// =============================================================================
// Version_Recipe - 05_RecipeHandler.scl
// Recipe-based motion handler with pre-scan validation
// No string parsing - direct array access for maximum efficiency
// =============================================================================

// -----------------------------------------------------------------------------
// FB_RecipeLoader - Copy the selected recipe from LOAD memory into work memory
// DOC:
//  purpose: DB_RecipeProgram1..PROGRAM_COUNT live in load memory (UNLINKED) and cannot be
//           read by the program directly. This FB copies the selected one into
//           "DB_SelectedRecipe" using TWO sequential READ_DBL sub-reference
//           transfers -- .Header first, then .Lines. Never the whole-DB form;
//           see "TWO TRANSFERS, NOT ONE" below for what that cost on the machine.
//           Runs once per cycle start, in STATE_RECIPE_LOAD(11), before the
//           pre-scan -- the machine is stationary and nothing else is pending.
//  inputs:  Execute (rising edge), ProgramNo (1..PROGRAM_COUNT), Reset (level)
//  outputs: Done, Busy, Error + ErrorCode, LoadedProgram
//  design:  Program/docs/LOADMEM_COPY_ON_SELECT.md  (gate-tested 2026-08-04)
//
//  READ_DBL call form -- both of these cost a build if you get them wrong:
//    * READ_DBL is an INSTANCE-LESS system function (SFC 83 heritage). Declaring
//      it as a multi-instance gives "Data type READ_DBL is unknown".
//    * RET_VAL is the FUNCTION RETURN VALUE, not an output parameter. Passing
//      it as RET_VAL => x gives "The formal parameter 'RET_VAL' is invalid".
//
//  TWO TRANSFERS, NOT ONE (changed 2026-08-06 after a field failure).
//  The first version copied the WHOLE DB in one call (SRCBLK := "DB_RecipeProgramN").
//  On the machine that delivered the Header correctly and left Lines completely
//  zero, with no error anywhere -- a structured copy that matched the first
//  member and gave up on the second. Re-reading the gate-test results
//  (loadmem_gatetest/result.md) shows why it was never caught: whole-DB mode was
//  only ever proven at 350 lines / 4.3 KB, while the 12 KB / 1000-line case was
//  proven with the SUB-REFERENCE form (SRCBLK := "...".Lines). Production ran the
//  one combination -- whole DB at 12 KB -- that no test covered.
//  So: Header and Lines are now copied in two sequential calls, each in the exact
//  form the gate test passed. A length or type mismatch on Lines surfaces as a
//  non-zero RET_VAL instead of a silently empty buffer.
//
//  THE SPLIT WAS NOT ENOUGH (2026-08-13, second field failure, same signature).
//  The claim that a sub-reference copy "cannot half-succeed" was wrong. On the
//  machine the .Lines call again returned RET_VAL = 0 with BUSY = FALSE while the
//  array stayed zero -- pre-scan caught it as 16#0313. RET_VAL/BUSY report that the
//  instruction accepted and closed the job, not that 12 KB of flash arrived, and
//  the moment this FB left ST_WAIT_LINES it dropped REQ and abandoned whatever was
//  still in flight. PLCSIM never reproduced it (host RAM, copy done in one call).
//  ST_WAIT_LINES therefore no longer trusts BUSY alone: it VERIFIES the copy and
//  re-issues the transfer up to LINES_RETRY_MAX times before failing. Do not
//  "simplify" that check away -- it is the only thing standing between a silent
//  partial copy and a machined part.
//
//  WHY THE VERIFY PROBES THE WHOLE ARRAY AND NOT JUST THE END MARKER.
//  Same day, with a 999-line recipe: the operator found DB_SelectedRecipe zero up
//  to roughly line 900 and CORRECT after it. The copy is not all-or-nothing, it is
//  PARTIAL -- and the part that landed is where the END marker lives, so a
//  marker-only test would have passed that buffer and the machine would have run
//  ~900 zero lines (X=0, Z=0) with the HMI counting up. That is exactly what
//  happened before this check existed. Five sampled probes replaced the marker
//  test, and chunking replaced the samples: at CHUNK_LINES = 100 EVERY line of the
//  staging buffer is poisoned and checked, so coverage is complete rather than
//  statistical. The 38-line case is the same fault seen from the other end: there
//  the marker sits at index 37, in the region that did NOT land, so pre-scan
//  caught it as 16#0313.
//  ErrorPhase says what failed: 1 = Header, 2 = chunk transfer, 3 = chunk verify.
//
//  WHAT THE VERIFY STILL CANNOT SEE, AND THE CHECKSUM (2026-08-14).
//  Poisoning proves every line was WRITTEN. It says nothing about whether the
//  right data arrived: a stale flash image, chunks reassembled at the wrong
//  stride, or a Header paired with another export's Lines all pass it, because
//  in every one of those cases all 1000 lines are written. So the loader now
//  folds an order-sensitive checksum over CMD + Param + F into ST_CHUNK_COPY
//  (the loop that already walks every line -- four adds per line, no second
//  pass) and compares it with Header.Checksum after the last chunk. Mismatch =
//  16#0316, ErrorPhase 4. Header.ProvidesChecksum = FALSE skips the check so
//  pre-2026-08-14 exports still load; that is deliberate, not a hole to close.
//  X and Z are NOT in the sum -- float32 on the CPU against float64 in the CAM
//  would eventually disagree on a VALID recipe, and an alarm that cries wolf is
//  worse than no alarm. Spec both sides build to:
//  Program/docs/letter_spinningcam_recipe_checksum.md
//
//  READING A FAILED LOAD (2026-08-14). ST_LATCH poisons every CMD in
//  DB_SelectedRecipe.Lines with 16#FF before the first transfer, so after a
//  failure the buffer says which chunks got in: 16#FF = never copied, 0 = copied
//  and the source is zero there, valid CMD = copied intact. ErrorChunk names the
//  chunk that ran out of retries; the poison shows what surrounds it.
//
//  THE SELECTION LATCH -- the one genuinely dangerous thing in this block.
//  READ_DBL is asynchronous and spans several scans with REQ held. SRCBLK is a
//  VARIANT and the S7-1200 cannot index a DB dynamically, so the source is
//  chosen by a CASE. If that CASE branch changed mid-transfer, the buffer would
//  receive the front of one recipe and the tail of another -- with RET_VAL = 0
//  and no error anywhere. The operator would machine a part that exists in no
//  recipe. Hence #selLatched: the branch is frozen at ST_LATCH and the live
//  ProgramNo input is ignored until the transfer completes.
//
//  Reset path: REQ is derived from the state EVERY scan and is never latched
//  independently, so there is no way for a transfer to stay in flight across a
//  reset, an E-Stop or an error acknowledge.
// -----------------------------------------------------------------------------
FUNCTION_BLOCK "FB_RecipeLoader"
{ S7_Optimized_Access := 'TRUE' }
VERSION : 0.3
    VAR_INPUT
        Execute   : Bool;           // Rising edge starts the copy
        ProgramNo : Int;            // 1..PROGRAM_COUNT -- which recipe to load
        Reset     : Bool;           // Level: abort, clear error, invalidate buffer
    END_VAR
    VAR_OUTPUT
        Done          : Bool;       // Copy complete AND verified, DB_SelectedRecipe is valid
        Busy          : Bool;       // Transfer in flight
        Error         : Bool;       // Copy failed -- FB_Process raises 16#0312 or 16#0314
        ErrorCode     : Word;       // READ_DBL RET_VAL, latched. Two sentinels that are
                                    // NOT RET_VAL values: 16#FFFF = watchdog timeout,
                                    // 16#0314 = a chunk never arrived intact
        ErrorPhase    : Int;        // 1 = Header transfer, 2 = chunk transfer (RET_VAL),
                                    // 3 = chunk verify (RET_VAL said OK, data did not arrive),
                                    // 4 = checksum mismatch (it all arrived, but it is not
                                    //     the recipe the CAM exported)
        ErrorChunk    : Int;        // Which chunk failed (1..CHUNK_COUNT), 0 = Header or
                                    // the assembled-buffer end-marker check
        RetryTotal    : Int;        // Re-issued transfers across the WHOLE load, cleared
                                    // at ST_LATCH. This is the margin gauge: a load that
                                    // succeeds with RetryTotal = 0 is comfortable; one
                                    // that succeeds with RetryTotal > 0 got there on
                                    // second attempts and CHUNK_LINES is too close to
                                    // whatever this CPU can actually deliver. Watch it on
                                    // the first hardware run -- a clean Done tells you
                                    // nothing on its own.
        LoadedProgram : Int;        // Which recipe is in the buffer (0 = none/invalid)
        ChecksumCalc  : UDInt;      // What WE computed over the reassembled buffer. On a
                                    // 16#0316 this is the number to compare against
                                    // DB_SelectedRecipe.Header.Checksum by hand -- and to
                                    // quote to the CAM developer, because one of the two
                                    // implementations is wrong and the pair says which.
        ChecksumOK    : Bool;       // TRUE = checked and matched. FALSE also means "the
                                    // recipe carries no checksum", so it is NOT a fault
                                    // indicator on its own -- read it with ProvidesChecksum.
    END_VAR
    VAR
        // READ_DBL is NOT declared here -- see the note above.
        tonWatch    : TON;          // Hang watchdog (RecipeLoadTimeout), per transfer
        state       : Int;          // see the ST_* constants below
        selLatched  : Int := 1;     // Frozen program number for the whole load.
                                    // Never cleared: keeps the instruction being
                                    // called with REQ=FALSE so it resets cleanly.
        chunkPhase  : Int;          // 0 = Header is the live call, 1..CHUNK_COUNT = that
                                    // chunk. Latched like selLatched: only ever changed
                                    // where REQ is already low, never mid-transfer.
        chunkRetry  : Int;          // Attempts already re-issued for the CURRENT chunk
        reqActive   : Bool;         // REQ level, derived from state every scan
        busyRaw     : Bool;         // READ_DBL BUSY
        retValRaw   : Int;          // READ_DBL return value (raw, every scan)
        chunkOK     : Bool;         // every line of the staging buffer came back written
        hdrLines    : Int;          // Header.LineCount, latched at ST_HDR_SETTLE. Used by
                                    // the checksum fold and the END-marker check, so it is
                                    // read ONCE from the Header and not re-read per chunk.
        dstBase     : Int;          // first DB_SelectedRecipe index of the current chunk
        sumA        : UDInt;        // checksum accumulator: running line sum
        sumB        : UDInt;        // checksum accumulator: sum of sumA -> order-sensitive
        prevExecute : Bool;
        rtExecute   : Bool;
    END_VAR
    VAR_TEMP
        i           : Int;          // loop index (poison / verify / copy)
        gLine       : Int;          // global recipe line index during the copy
    END_VAR
    CONST
        ST_IDLE        : Int := 0;
        ST_LATCH       : Int := 10;
        ST_REQ_HDR     : Int := 20;  // Header transfer
        ST_WAIT_HDR    : Int := 30;
        ST_HDR_SETTLE  : Int := 35;  // One scan with REQ low so the Header call sees
                                     // its job closed before the CASE switches
        ST_CHUNK_PREP  : Int := 38;  // REQ low: poison the staging buffer, then request.
                                     // Also the settle scan BETWEEN chunks and the
                                     // re-poison step before a retry.
        ST_REQ_CHUNK   : Int := 40;
        ST_WAIT_CHUNK  : Int := 50;
        ST_CHUNK_COPY  : Int := 57;  // staging -> DB_SelectedRecipe (work memory, sync)
        ST_DONE        : Int := 60;
        ST_ERROR       : Int := 90;
        CHUNK_RETRY_MAX : Int := 3;  // re-issues per chunk before 16#0314. Each attempt
                                     // is bounded by RecipeLoadTimeout.
        CMD_PROGRAM_END : Int := 99; // Mandatory last-line marker (PLC_Recipe_Format_Spec.md)
        POISON_CMD     : Int := 255; // 16#FF -- no recipe CMD can be this value
        // Chunk geometry. COUPLED to tools/gen_recipe_slots.py (CHUNK_LINES /
        // CHUNK_COUNT) and to the DB_RecipeProgram*.Lines1..N declarations it
        // emits. Change them together or the transfers go out of step.
        // <<< GENERATED:CHUNK_GEOMETRY -- do not hand-edit; run tools/gen_recipe_slots.py >>>
        CHUNK_LINES    : Int := 100;
        CHUNK_COUNT    : Int := 8;
        LINES_MAX      : Int := 800; // = CHUNK_LINES * CHUNK_COUNT, and the bound of
                                      // DB_SelectedRecipe.Lines + the pre-scan guard
        // <<< END GENERATED:CHUNK_GEOMETRY >>>
        // <<< GENERATED:PROGRAM_COUNT -- do not hand-edit; run tools/gen_recipe_slots.py >>>
        PROGRAM_COUNT : Int := 10;  // Slot count. Generated -- must match the DB_RecipeProgram* count.
        // <<< END GENERATED:PROGRAM_COUNT >>>
    END_CONST
BEGIN
    // -------------------------------------------------------------------------
    // Rising edge on Execute
    // -------------------------------------------------------------------------
    #rtExecute := #Execute AND NOT #prevExecute;
    #prevExecute := #Execute;

    // -------------------------------------------------------------------------
    // Reset -- always honoured. Drives REQ low via the state on the next line.
    // -------------------------------------------------------------------------
    IF #Reset THEN
        #state := ST_IDLE;
        #Done := FALSE;
        #Error := FALSE;
        #ErrorCode := 16#0000;
        #ErrorPhase := 0;
        #ErrorChunk := 0;
        #chunkPhase := 0;           // idle on the Header branch, REQ low
        #chunkRetry := 0;
        #RetryTotal := 0;
        #LoadedProgram := 0;        // Buffer is no longer trusted -> forces a re-load
        #ChecksumCalc := 0;
        #ChecksumOK := FALSE;
    END_IF;

    // -------------------------------------------------------------------------
    // REQ is derived from state EVERY SCAN -- never latched on its own.
    // ST_CHUNK_PREP is deliberately excluded: that is the scan where the previous
    // job is closed, the staging buffer is poisoned and the watchdog resets.
    // -------------------------------------------------------------------------
    #reqActive := (#state = ST_REQ_HDR) OR (#state = ST_WAIT_HDR)
                  OR (#state = ST_REQ_CHUNK) OR (#state = ST_WAIT_CHUNK);

    // -------------------------------------------------------------------------
    // THE READ_DBL CALL BLOCK
    // Outer CASE = which recipe (#selLatched), inner CASE = which transfer
    // (#chunkPhase: 0 = Header, 1..CHUNK_COUNT = Lines chunks). Exactly ONE call
    // executes per scan. Both selectors are latched, never the live inputs.
    // -------------------------------------------------------------------------
    // <<< GENERATED:LOADER_CASE -- do not hand-edit; run tools/gen_recipe_slots.py >>>
    CASE #selLatched OF
        1:  CASE #chunkPhase OF
                0: #retValRaw := READ_DBL(REQ := #reqActive, SRCBLK := "DB_RecipeProgram1".Header,
                                           BUSY => #busyRaw, DSTBLK := "DB_SelectedRecipe".Header);
                1: #retValRaw := READ_DBL(REQ := #reqActive, SRCBLK := "DB_RecipeProgram1".Lines1,
                                           BUSY => #busyRaw, DSTBLK := "DB_RecipeChunk".Lines);
                2: #retValRaw := READ_DBL(REQ := #reqActive, SRCBLK := "DB_RecipeProgram1".Lines2,
                                           BUSY => #busyRaw, DSTBLK := "DB_RecipeChunk".Lines);
                3: #retValRaw := READ_DBL(REQ := #reqActive, SRCBLK := "DB_RecipeProgram1".Lines3,
                                           BUSY => #busyRaw, DSTBLK := "DB_RecipeChunk".Lines);
                4: #retValRaw := READ_DBL(REQ := #reqActive, SRCBLK := "DB_RecipeProgram1".Lines4,
                                           BUSY => #busyRaw, DSTBLK := "DB_RecipeChunk".Lines);
                5: #retValRaw := READ_DBL(REQ := #reqActive, SRCBLK := "DB_RecipeProgram1".Lines5,
                                           BUSY => #busyRaw, DSTBLK := "DB_RecipeChunk".Lines);
                6: #retValRaw := READ_DBL(REQ := #reqActive, SRCBLK := "DB_RecipeProgram1".Lines6,
                                           BUSY => #busyRaw, DSTBLK := "DB_RecipeChunk".Lines);
                7: #retValRaw := READ_DBL(REQ := #reqActive, SRCBLK := "DB_RecipeProgram1".Lines7,
                                           BUSY => #busyRaw, DSTBLK := "DB_RecipeChunk".Lines);
                8: #retValRaw := READ_DBL(REQ := #reqActive, SRCBLK := "DB_RecipeProgram1".Lines8,
                                           BUSY => #busyRaw, DSTBLK := "DB_RecipeChunk".Lines);
            END_CASE;
        2:  CASE #chunkPhase OF
                0: #retValRaw := READ_DBL(REQ := #reqActive, SRCBLK := "DB_RecipeProgram2".Header,
                                           BUSY => #busyRaw, DSTBLK := "DB_SelectedRecipe".Header);
                1: #retValRaw := READ_DBL(REQ := #reqActive, SRCBLK := "DB_RecipeProgram2".Lines1,
                                           BUSY => #busyRaw, DSTBLK := "DB_RecipeChunk".Lines);
                2: #retValRaw := READ_DBL(REQ := #reqActive, SRCBLK := "DB_RecipeProgram2".Lines2,
                                           BUSY => #busyRaw, DSTBLK := "DB_RecipeChunk".Lines);
                3: #retValRaw := READ_DBL(REQ := #reqActive, SRCBLK := "DB_RecipeProgram2".Lines3,
                                           BUSY => #busyRaw, DSTBLK := "DB_RecipeChunk".Lines);
                4: #retValRaw := READ_DBL(REQ := #reqActive, SRCBLK := "DB_RecipeProgram2".Lines4,
                                           BUSY => #busyRaw, DSTBLK := "DB_RecipeChunk".Lines);
                5: #retValRaw := READ_DBL(REQ := #reqActive, SRCBLK := "DB_RecipeProgram2".Lines5,
                                           BUSY => #busyRaw, DSTBLK := "DB_RecipeChunk".Lines);
                6: #retValRaw := READ_DBL(REQ := #reqActive, SRCBLK := "DB_RecipeProgram2".Lines6,
                                           BUSY => #busyRaw, DSTBLK := "DB_RecipeChunk".Lines);
                7: #retValRaw := READ_DBL(REQ := #reqActive, SRCBLK := "DB_RecipeProgram2".Lines7,
                                           BUSY => #busyRaw, DSTBLK := "DB_RecipeChunk".Lines);
                8: #retValRaw := READ_DBL(REQ := #reqActive, SRCBLK := "DB_RecipeProgram2".Lines8,
                                           BUSY => #busyRaw, DSTBLK := "DB_RecipeChunk".Lines);
            END_CASE;
        3:  CASE #chunkPhase OF
                0: #retValRaw := READ_DBL(REQ := #reqActive, SRCBLK := "DB_RecipeProgram3".Header,
                                           BUSY => #busyRaw, DSTBLK := "DB_SelectedRecipe".Header);
                1: #retValRaw := READ_DBL(REQ := #reqActive, SRCBLK := "DB_RecipeProgram3".Lines1,
                                           BUSY => #busyRaw, DSTBLK := "DB_RecipeChunk".Lines);
                2: #retValRaw := READ_DBL(REQ := #reqActive, SRCBLK := "DB_RecipeProgram3".Lines2,
                                           BUSY => #busyRaw, DSTBLK := "DB_RecipeChunk".Lines);
                3: #retValRaw := READ_DBL(REQ := #reqActive, SRCBLK := "DB_RecipeProgram3".Lines3,
                                           BUSY => #busyRaw, DSTBLK := "DB_RecipeChunk".Lines);
                4: #retValRaw := READ_DBL(REQ := #reqActive, SRCBLK := "DB_RecipeProgram3".Lines4,
                                           BUSY => #busyRaw, DSTBLK := "DB_RecipeChunk".Lines);
                5: #retValRaw := READ_DBL(REQ := #reqActive, SRCBLK := "DB_RecipeProgram3".Lines5,
                                           BUSY => #busyRaw, DSTBLK := "DB_RecipeChunk".Lines);
                6: #retValRaw := READ_DBL(REQ := #reqActive, SRCBLK := "DB_RecipeProgram3".Lines6,
                                           BUSY => #busyRaw, DSTBLK := "DB_RecipeChunk".Lines);
                7: #retValRaw := READ_DBL(REQ := #reqActive, SRCBLK := "DB_RecipeProgram3".Lines7,
                                           BUSY => #busyRaw, DSTBLK := "DB_RecipeChunk".Lines);
                8: #retValRaw := READ_DBL(REQ := #reqActive, SRCBLK := "DB_RecipeProgram3".Lines8,
                                           BUSY => #busyRaw, DSTBLK := "DB_RecipeChunk".Lines);
            END_CASE;
        4:  CASE #chunkPhase OF
                0: #retValRaw := READ_DBL(REQ := #reqActive, SRCBLK := "DB_RecipeProgram4".Header,
                                           BUSY => #busyRaw, DSTBLK := "DB_SelectedRecipe".Header);
                1: #retValRaw := READ_DBL(REQ := #reqActive, SRCBLK := "DB_RecipeProgram4".Lines1,
                                           BUSY => #busyRaw, DSTBLK := "DB_RecipeChunk".Lines);
                2: #retValRaw := READ_DBL(REQ := #reqActive, SRCBLK := "DB_RecipeProgram4".Lines2,
                                           BUSY => #busyRaw, DSTBLK := "DB_RecipeChunk".Lines);
                3: #retValRaw := READ_DBL(REQ := #reqActive, SRCBLK := "DB_RecipeProgram4".Lines3,
                                           BUSY => #busyRaw, DSTBLK := "DB_RecipeChunk".Lines);
                4: #retValRaw := READ_DBL(REQ := #reqActive, SRCBLK := "DB_RecipeProgram4".Lines4,
                                           BUSY => #busyRaw, DSTBLK := "DB_RecipeChunk".Lines);
                5: #retValRaw := READ_DBL(REQ := #reqActive, SRCBLK := "DB_RecipeProgram4".Lines5,
                                           BUSY => #busyRaw, DSTBLK := "DB_RecipeChunk".Lines);
                6: #retValRaw := READ_DBL(REQ := #reqActive, SRCBLK := "DB_RecipeProgram4".Lines6,
                                           BUSY => #busyRaw, DSTBLK := "DB_RecipeChunk".Lines);
                7: #retValRaw := READ_DBL(REQ := #reqActive, SRCBLK := "DB_RecipeProgram4".Lines7,
                                           BUSY => #busyRaw, DSTBLK := "DB_RecipeChunk".Lines);
                8: #retValRaw := READ_DBL(REQ := #reqActive, SRCBLK := "DB_RecipeProgram4".Lines8,
                                           BUSY => #busyRaw, DSTBLK := "DB_RecipeChunk".Lines);
            END_CASE;
        5:  CASE #chunkPhase OF
                0: #retValRaw := READ_DBL(REQ := #reqActive, SRCBLK := "DB_RecipeProgram5".Header,
                                           BUSY => #busyRaw, DSTBLK := "DB_SelectedRecipe".Header);
                1: #retValRaw := READ_DBL(REQ := #reqActive, SRCBLK := "DB_RecipeProgram5".Lines1,
                                           BUSY => #busyRaw, DSTBLK := "DB_RecipeChunk".Lines);
                2: #retValRaw := READ_DBL(REQ := #reqActive, SRCBLK := "DB_RecipeProgram5".Lines2,
                                           BUSY => #busyRaw, DSTBLK := "DB_RecipeChunk".Lines);
                3: #retValRaw := READ_DBL(REQ := #reqActive, SRCBLK := "DB_RecipeProgram5".Lines3,
                                           BUSY => #busyRaw, DSTBLK := "DB_RecipeChunk".Lines);
                4: #retValRaw := READ_DBL(REQ := #reqActive, SRCBLK := "DB_RecipeProgram5".Lines4,
                                           BUSY => #busyRaw, DSTBLK := "DB_RecipeChunk".Lines);
                5: #retValRaw := READ_DBL(REQ := #reqActive, SRCBLK := "DB_RecipeProgram5".Lines5,
                                           BUSY => #busyRaw, DSTBLK := "DB_RecipeChunk".Lines);
                6: #retValRaw := READ_DBL(REQ := #reqActive, SRCBLK := "DB_RecipeProgram5".Lines6,
                                           BUSY => #busyRaw, DSTBLK := "DB_RecipeChunk".Lines);
                7: #retValRaw := READ_DBL(REQ := #reqActive, SRCBLK := "DB_RecipeProgram5".Lines7,
                                           BUSY => #busyRaw, DSTBLK := "DB_RecipeChunk".Lines);
                8: #retValRaw := READ_DBL(REQ := #reqActive, SRCBLK := "DB_RecipeProgram5".Lines8,
                                           BUSY => #busyRaw, DSTBLK := "DB_RecipeChunk".Lines);
            END_CASE;
        6:  CASE #chunkPhase OF
                0: #retValRaw := READ_DBL(REQ := #reqActive, SRCBLK := "DB_RecipeProgram6".Header,
                                           BUSY => #busyRaw, DSTBLK := "DB_SelectedRecipe".Header);
                1: #retValRaw := READ_DBL(REQ := #reqActive, SRCBLK := "DB_RecipeProgram6".Lines1,
                                           BUSY => #busyRaw, DSTBLK := "DB_RecipeChunk".Lines);
                2: #retValRaw := READ_DBL(REQ := #reqActive, SRCBLK := "DB_RecipeProgram6".Lines2,
                                           BUSY => #busyRaw, DSTBLK := "DB_RecipeChunk".Lines);
                3: #retValRaw := READ_DBL(REQ := #reqActive, SRCBLK := "DB_RecipeProgram6".Lines3,
                                           BUSY => #busyRaw, DSTBLK := "DB_RecipeChunk".Lines);
                4: #retValRaw := READ_DBL(REQ := #reqActive, SRCBLK := "DB_RecipeProgram6".Lines4,
                                           BUSY => #busyRaw, DSTBLK := "DB_RecipeChunk".Lines);
                5: #retValRaw := READ_DBL(REQ := #reqActive, SRCBLK := "DB_RecipeProgram6".Lines5,
                                           BUSY => #busyRaw, DSTBLK := "DB_RecipeChunk".Lines);
                6: #retValRaw := READ_DBL(REQ := #reqActive, SRCBLK := "DB_RecipeProgram6".Lines6,
                                           BUSY => #busyRaw, DSTBLK := "DB_RecipeChunk".Lines);
                7: #retValRaw := READ_DBL(REQ := #reqActive, SRCBLK := "DB_RecipeProgram6".Lines7,
                                           BUSY => #busyRaw, DSTBLK := "DB_RecipeChunk".Lines);
                8: #retValRaw := READ_DBL(REQ := #reqActive, SRCBLK := "DB_RecipeProgram6".Lines8,
                                           BUSY => #busyRaw, DSTBLK := "DB_RecipeChunk".Lines);
            END_CASE;
        7:  CASE #chunkPhase OF
                0: #retValRaw := READ_DBL(REQ := #reqActive, SRCBLK := "DB_RecipeProgram7".Header,
                                           BUSY => #busyRaw, DSTBLK := "DB_SelectedRecipe".Header);
                1: #retValRaw := READ_DBL(REQ := #reqActive, SRCBLK := "DB_RecipeProgram7".Lines1,
                                           BUSY => #busyRaw, DSTBLK := "DB_RecipeChunk".Lines);
                2: #retValRaw := READ_DBL(REQ := #reqActive, SRCBLK := "DB_RecipeProgram7".Lines2,
                                           BUSY => #busyRaw, DSTBLK := "DB_RecipeChunk".Lines);
                3: #retValRaw := READ_DBL(REQ := #reqActive, SRCBLK := "DB_RecipeProgram7".Lines3,
                                           BUSY => #busyRaw, DSTBLK := "DB_RecipeChunk".Lines);
                4: #retValRaw := READ_DBL(REQ := #reqActive, SRCBLK := "DB_RecipeProgram7".Lines4,
                                           BUSY => #busyRaw, DSTBLK := "DB_RecipeChunk".Lines);
                5: #retValRaw := READ_DBL(REQ := #reqActive, SRCBLK := "DB_RecipeProgram7".Lines5,
                                           BUSY => #busyRaw, DSTBLK := "DB_RecipeChunk".Lines);
                6: #retValRaw := READ_DBL(REQ := #reqActive, SRCBLK := "DB_RecipeProgram7".Lines6,
                                           BUSY => #busyRaw, DSTBLK := "DB_RecipeChunk".Lines);
                7: #retValRaw := READ_DBL(REQ := #reqActive, SRCBLK := "DB_RecipeProgram7".Lines7,
                                           BUSY => #busyRaw, DSTBLK := "DB_RecipeChunk".Lines);
                8: #retValRaw := READ_DBL(REQ := #reqActive, SRCBLK := "DB_RecipeProgram7".Lines8,
                                           BUSY => #busyRaw, DSTBLK := "DB_RecipeChunk".Lines);
            END_CASE;
        8:  CASE #chunkPhase OF
                0: #retValRaw := READ_DBL(REQ := #reqActive, SRCBLK := "DB_RecipeProgram8".Header,
                                           BUSY => #busyRaw, DSTBLK := "DB_SelectedRecipe".Header);
                1: #retValRaw := READ_DBL(REQ := #reqActive, SRCBLK := "DB_RecipeProgram8".Lines1,
                                           BUSY => #busyRaw, DSTBLK := "DB_RecipeChunk".Lines);
                2: #retValRaw := READ_DBL(REQ := #reqActive, SRCBLK := "DB_RecipeProgram8".Lines2,
                                           BUSY => #busyRaw, DSTBLK := "DB_RecipeChunk".Lines);
                3: #retValRaw := READ_DBL(REQ := #reqActive, SRCBLK := "DB_RecipeProgram8".Lines3,
                                           BUSY => #busyRaw, DSTBLK := "DB_RecipeChunk".Lines);
                4: #retValRaw := READ_DBL(REQ := #reqActive, SRCBLK := "DB_RecipeProgram8".Lines4,
                                           BUSY => #busyRaw, DSTBLK := "DB_RecipeChunk".Lines);
                5: #retValRaw := READ_DBL(REQ := #reqActive, SRCBLK := "DB_RecipeProgram8".Lines5,
                                           BUSY => #busyRaw, DSTBLK := "DB_RecipeChunk".Lines);
                6: #retValRaw := READ_DBL(REQ := #reqActive, SRCBLK := "DB_RecipeProgram8".Lines6,
                                           BUSY => #busyRaw, DSTBLK := "DB_RecipeChunk".Lines);
                7: #retValRaw := READ_DBL(REQ := #reqActive, SRCBLK := "DB_RecipeProgram8".Lines7,
                                           BUSY => #busyRaw, DSTBLK := "DB_RecipeChunk".Lines);
                8: #retValRaw := READ_DBL(REQ := #reqActive, SRCBLK := "DB_RecipeProgram8".Lines8,
                                           BUSY => #busyRaw, DSTBLK := "DB_RecipeChunk".Lines);
            END_CASE;
        9:  CASE #chunkPhase OF
                0: #retValRaw := READ_DBL(REQ := #reqActive, SRCBLK := "DB_RecipeProgram9".Header,
                                           BUSY => #busyRaw, DSTBLK := "DB_SelectedRecipe".Header);
                1: #retValRaw := READ_DBL(REQ := #reqActive, SRCBLK := "DB_RecipeProgram9".Lines1,
                                           BUSY => #busyRaw, DSTBLK := "DB_RecipeChunk".Lines);
                2: #retValRaw := READ_DBL(REQ := #reqActive, SRCBLK := "DB_RecipeProgram9".Lines2,
                                           BUSY => #busyRaw, DSTBLK := "DB_RecipeChunk".Lines);
                3: #retValRaw := READ_DBL(REQ := #reqActive, SRCBLK := "DB_RecipeProgram9".Lines3,
                                           BUSY => #busyRaw, DSTBLK := "DB_RecipeChunk".Lines);
                4: #retValRaw := READ_DBL(REQ := #reqActive, SRCBLK := "DB_RecipeProgram9".Lines4,
                                           BUSY => #busyRaw, DSTBLK := "DB_RecipeChunk".Lines);
                5: #retValRaw := READ_DBL(REQ := #reqActive, SRCBLK := "DB_RecipeProgram9".Lines5,
                                           BUSY => #busyRaw, DSTBLK := "DB_RecipeChunk".Lines);
                6: #retValRaw := READ_DBL(REQ := #reqActive, SRCBLK := "DB_RecipeProgram9".Lines6,
                                           BUSY => #busyRaw, DSTBLK := "DB_RecipeChunk".Lines);
                7: #retValRaw := READ_DBL(REQ := #reqActive, SRCBLK := "DB_RecipeProgram9".Lines7,
                                           BUSY => #busyRaw, DSTBLK := "DB_RecipeChunk".Lines);
                8: #retValRaw := READ_DBL(REQ := #reqActive, SRCBLK := "DB_RecipeProgram9".Lines8,
                                           BUSY => #busyRaw, DSTBLK := "DB_RecipeChunk".Lines);
            END_CASE;
        10: CASE #chunkPhase OF
                0: #retValRaw := READ_DBL(REQ := #reqActive, SRCBLK := "DB_RecipeProgram10".Header,
                                           BUSY => #busyRaw, DSTBLK := "DB_SelectedRecipe".Header);
                1: #retValRaw := READ_DBL(REQ := #reqActive, SRCBLK := "DB_RecipeProgram10".Lines1,
                                           BUSY => #busyRaw, DSTBLK := "DB_RecipeChunk".Lines);
                2: #retValRaw := READ_DBL(REQ := #reqActive, SRCBLK := "DB_RecipeProgram10".Lines2,
                                           BUSY => #busyRaw, DSTBLK := "DB_RecipeChunk".Lines);
                3: #retValRaw := READ_DBL(REQ := #reqActive, SRCBLK := "DB_RecipeProgram10".Lines3,
                                           BUSY => #busyRaw, DSTBLK := "DB_RecipeChunk".Lines);
                4: #retValRaw := READ_DBL(REQ := #reqActive, SRCBLK := "DB_RecipeProgram10".Lines4,
                                           BUSY => #busyRaw, DSTBLK := "DB_RecipeChunk".Lines);
                5: #retValRaw := READ_DBL(REQ := #reqActive, SRCBLK := "DB_RecipeProgram10".Lines5,
                                           BUSY => #busyRaw, DSTBLK := "DB_RecipeChunk".Lines);
                6: #retValRaw := READ_DBL(REQ := #reqActive, SRCBLK := "DB_RecipeProgram10".Lines6,
                                           BUSY => #busyRaw, DSTBLK := "DB_RecipeChunk".Lines);
                7: #retValRaw := READ_DBL(REQ := #reqActive, SRCBLK := "DB_RecipeProgram10".Lines7,
                                           BUSY => #busyRaw, DSTBLK := "DB_RecipeChunk".Lines);
                8: #retValRaw := READ_DBL(REQ := #reqActive, SRCBLK := "DB_RecipeProgram10".Lines8,
                                           BUSY => #busyRaw, DSTBLK := "DB_RecipeChunk".Lines);
            END_CASE;
    END_CASE;
    // <<< END GENERATED:LOADER_CASE >>>

    // -------------------------------------------------------------------------
    // Hang watchdog -- only runs while a transfer is in flight
    // -------------------------------------------------------------------------
    #tonWatch(IN := #reqActive, PT := "DB_MachineConfig".RecipeLoadTimeout);

    // -------------------------------------------------------------------------
    // State machine
    // -------------------------------------------------------------------------
    CASE #state OF

        // === ST_IDLE (0) ===
        ST_IDLE:
            IF #rtExecute AND #ProgramNo >= 1 AND #ProgramNo <= PROGRAM_COUNT THEN
                #state := ST_LATCH;
            END_IF;

        // === ST_LATCH (10) -- freeze the selection, poison the header ===
        ST_LATCH:
            #selLatched := #ProgramNo;      // the latch. Everything downstream uses this.
            #chunkPhase := 0;               // always start with the Header transfer
            #chunkRetry := 0;
            #Done := FALSE;
            #Error := FALSE;
            #ErrorCode := 16#0000;
            #ErrorPhase := 0;
            #ErrorChunk := 0;
            #RetryTotal := 0;               // margin gauge, per load
            #LoadedProgram := 0;            // buffer invalid until the copy lands
            #sumA := 0;                     // checksum accumulators, per load
            #sumB := 0;
            #ChecksumCalc := 0;
            #ChecksumOK := FALSE;
            // POISON (2026-08-06): a failed load must leave a buffer that CANNOT
            // pass pre-scan. DB_SelectedRecipe survives delta downloads and failed
            // transfers, so header data from an OLD copy would otherwise sit there
            // looking like evidence that "the copy worked".
            "DB_SelectedRecipe".Header.LineCount := 0;
            "DB_SelectedRecipe".Header.sName := '';
            "DB_SelectedRecipe".Header.Valid := FALSE;

            // POISON THE DESTINATION TOO (2026-08-14). Not needed for safety --
            // every chunk is verified in the staging buffer before it is allowed
            // in here, and CHUNK_LINES * CHUNK_COUNT covers the whole array, so
            // nothing stale can survive a COMPLETE load. It is here for the two
            // cases where that is not enough:
            //   * DIAGNOSIS. After a failed load the buffer is a map: 16#FF = that
            //     chunk never arrived, 0 = it arrived and the source is genuinely
            //     zero there, a valid CMD = it arrived intact. Clearing to ZERO
            //     instead would destroy exactly that distinction -- a hole and a
            //     legitimately-zero line would look identical, which is what made
            //     the 999-line failure so hard to read in the first place.
            //   * FULL-COVERAGE IS AN INVARIANT, NOT A GUARANTEE. "No stale data"
            //     currently rests on CHUNK_LINES * CHUNK_COUNT = LINES_MAX. Retune
            //     the geometry to something that does not cover the array and the
            //     tail would quietly keep the PREVIOUS recipe. With this loop it
            //     keeps 16#FF instead, and pre-scan/the end-marker check trip.
            // ~1000 byte writes in one scan, at cycle start, machine stationary,
            // nothing else pending -- measured against RecipeLoadTimeout, not the
            // motion loop. Do not move it into the per-chunk path to "spread the
            // cost": it must run ONCE, before the first transfer, or a retry would
            // wipe chunks that already landed.
            FOR #i := 0 TO LINES_MAX - 1 DO
                "DB_SelectedRecipe".Lines[#i].CMD := 16#FF;
            END_FOR;
            #state := ST_REQ_HDR;

        // === ST_REQ_HDR (20) -- first scan with REQ high, Header branch ===
        ST_REQ_HDR:
            #state := ST_WAIT_HDR;

        // === ST_WAIT_HDR (30) -- hold REQ on the SAME branch until BUSY drops ===
        // ErrorCode is LATCHED here, not mirrored every scan: once REQ falls the
        // next call returns its idle value and would wipe the real result.
        ST_WAIT_HDR:
            IF #tonWatch.Q THEN
                #ErrorCode := 16#FFFF;      // watchdog: BUSY never cleared
                #ErrorPhase := 1;
                #state := ST_ERROR;
            ELSIF NOT #busyRaw THEN
                IF #retValRaw = 0 THEN
                    #state := ST_HDR_SETTLE;
                ELSE
                    #ErrorCode := INT_TO_WORD(#retValRaw);
                    #ErrorPhase := 1;
                    #state := ST_ERROR;
                END_IF;
            END_IF;

        // === ST_HDR_SETTLE (35) -- one scan with REQ low, then start chunk 1 ===
        // The Header has landed, so LineCount is known before the first chunk.
        // Latch it here: the checksum fold needs it per line, and re-reading the
        // Header 1000 times would make a moving target of the bound.
        ST_HDR_SETTLE:
            #hdrLines := "DB_SelectedRecipe".Header.LineCount;
            #chunkPhase := 1;
            #chunkRetry := 0;
            #state := ST_CHUNK_PREP;

        // === ST_CHUNK_PREP (38) -- REQ low: poison the staging buffer ===
        // Every line gets 16#FF in its CMD byte. After the transfer, ANY line
        // still holding 16#FF proves that line was never written. At CHUNK_LINES
        // = 100 this is complete coverage, not a sample: the scattered holes seen
        // on the machine (data around line 200 on one attempt, past 850 on
        // another) cannot slip through it.
        ST_CHUNK_PREP:
            FOR #i := 0 TO CHUNK_LINES - 1 DO
                "DB_RecipeChunk".Lines[#i].CMD := 16#FF;
            END_FOR;
            #state := ST_REQ_CHUNK;

        // === ST_REQ_CHUNK (40) -- first scan with REQ high on this chunk ===
        ST_REQ_CHUNK:
            #state := ST_WAIT_CHUNK;

        // === ST_WAIT_CHUNK (50) -- wait, then VERIFY before believing it ===
        // BUSY = FALSE with RET_VAL = 0 reports that the instruction closed the
        // job, NOT that the bytes arrived. That distinction is the entire bug.
        ST_WAIT_CHUNK:
            IF #tonWatch.Q THEN
                #ErrorCode := 16#FFFF;
                #ErrorPhase := 2;
                #ErrorChunk := #chunkPhase;
                #state := ST_ERROR;
            ELSIF NOT #busyRaw THEN
                IF #retValRaw <> 0 THEN
                    #ErrorCode := INT_TO_WORD(#retValRaw);
                    #ErrorPhase := 2;
                    #ErrorChunk := #chunkPhase;
                    #state := ST_ERROR;
                ELSE
                    #chunkOK := TRUE;
                    FOR #i := 0 TO CHUNK_LINES - 1 DO
                        IF BYTE_TO_INT("DB_RecipeChunk".Lines[#i].CMD) = POISON_CMD THEN
                            #chunkOK := FALSE;
                        END_IF;
                    END_FOR;

                    IF #chunkOK THEN
                        #state := ST_CHUNK_COPY;
                    ELSIF #chunkRetry < CHUNK_RETRY_MAX THEN
                        #chunkRetry := #chunkRetry + 1;
                        #RetryTotal := #RetryTotal + 1;
                        #state := ST_CHUNK_PREP;    // re-poison and re-issue THIS chunk
                    ELSE
                        // Out of attempts on this chunk. Not a READ_DBL failure --
                        // it claimed success every time -- so it gets its own code.
                        #ErrorCode := 16#0314;
                        #ErrorPhase := 3;
                        #ErrorChunk := #chunkPhase;
                        #state := ST_ERROR;
                    END_IF;
                END_IF;
            END_IF;

        // === ST_CHUNK_COPY (57) -- staging -> DB_SelectedRecipe ===
        // Work memory to work memory, synchronous, one scan. Variable indices are
        // legal here; it is only the READ_DBL VARIANT that must be constant.
        // The checksum is folded into THIS loop rather than run as a separate pass
        // over 1000 lines: the loop already touches every line, so the cost is four
        // adds per line instead of a second traversal. Each chunk reaches here
        // exactly once -- a failed verify retries from ST_CHUNK_PREP and never
        // copies -- so no line can be accumulated twice.
        ST_CHUNK_COPY:
            #dstBase := (#chunkPhase - 1) * CHUNK_LINES;
            FOR #i := 0 TO CHUNK_LINES - 1 DO
                "DB_SelectedRecipe".Lines[#dstBase + #i] := "DB_RecipeChunk".Lines[#i];

                // Only the EMITTED lines count. Everything from LineCount to 999 is
                // padding the CAM never wrote and must not enter the sum, or the two
                // sides would have to agree on padding as well as on data.
                #gLine := #dstBase + #i;
                IF #gLine < #hdrLines THEN
                    // F goes in as its unsigned 16-bit BIT PATTERN, not its value:
                    // INT_TO_UDINT of a negative Int is a conversion fault waiting for
                    // a malformed export, and this way both sides agree regardless of
                    // sign. CMD and Param are bytes, so they are always non-negative.
                    #sumA := #sumA
                             + INT_TO_UDINT(BYTE_TO_INT("DB_RecipeChunk".Lines[#i].CMD)
                                            + BYTE_TO_INT("DB_RecipeChunk".Lines[#i].Param))
                             + DWORD_TO_UDINT(WORD_TO_DWORD(INT_TO_WORD("DB_RecipeChunk".Lines[#i].F)));
                    #sumB := #sumB + #sumA;     // running sum -> order-sensitive
                END_IF;
            END_FOR;

            IF #chunkPhase < CHUNK_COUNT THEN
                #chunkPhase := #chunkPhase + 1;
                #chunkRetry := 0;               // fresh budget for the next chunk
                #state := ST_CHUNK_PREP;
            ELSE
                // Last chunk in. Final cross-check: the recipe format guarantees
                // the last line is CMD = 99, so the assembled buffer must end
                // where the Header says it does. Catches a Header and a Lines set
                // that came from different states of the source DB.
                // #hdrLines was latched at ST_HDR_SETTLE -- do not re-read it here.
                //
                // CHECKSUM (2026-08-14). Seal the accumulators and compare against
                // the CAM's figure. This is the ONLY check that looks at the DATA
                // rather than at whether bytes were written: the poison verify
                // above proves every line arrived, not that the right recipe did.
                // It catches a stale flash image, chunks reassembled at the wrong
                // stride, and a Header paired with someone else's Lines.
                // XOR is a bit-string operation, hence the two conversions.
                #ChecksumCalc := DWORD_TO_UDINT(
                    UDINT_TO_DWORD(#sumB)
                    XOR UDINT_TO_DWORD(#sumA + INT_TO_UDINT(#hdrLines)));

                IF #hdrLines >= 1 AND #hdrLines <= LINES_MAX
                   AND BYTE_TO_INT("DB_SelectedRecipe".Lines[#hdrLines - 1].CMD) <> CMD_PROGRAM_END THEN
                    #ErrorCode := 16#0314;
                    #ErrorPhase := 3;
                    #ErrorChunk := 0;           // 0 = assembled buffer, not one chunk
                    #state := ST_ERROR;

                ELSIF "DB_SelectedRecipe".Header.ProvidesChecksum
                      AND #ChecksumCalc <> "DB_SelectedRecipe".Header.Checksum THEN
                    // Everything arrived and none of it is what was exported.
                    // Deliberately its own code: 16#0314 sends the operator looking
                    // for a transfer fault, and there is no transfer fault here.
                    #ErrorCode := 16#0316;
                    #ErrorPhase := 4;
                    #ErrorChunk := 0;
                    #state := ST_ERROR;

                ELSE
                    // Matched, or the recipe predates the field. ProvidesChecksum
                    // = FALSE is ACCEPTED on purpose -- making it mandatory would
                    // brick every existing export the moment this is downloaded.
                    #ChecksumOK := "DB_SelectedRecipe".Header.ProvidesChecksum;
                    #LoadedProgram := #selLatched;
                    #Done := TRUE;
                    #state := ST_DONE;
                END_IF;
            END_IF;

        // === ST_DONE (60) ===
        // Done stays TRUE so FB_Process can move on. A new rising edge re-loads,
        // which is what a program change or a restart must do.
        ST_DONE:
            #Done := TRUE;
            IF #rtExecute AND #ProgramNo >= 1 AND #ProgramNo <= PROGRAM_COUNT THEN
                #state := ST_LATCH;
            END_IF;

        // === ST_ERROR (90) -- cleared only by Reset ===
        ST_ERROR:
            #Error := TRUE;
            #Done := FALSE;
            #LoadedProgram := 0;
    END_CASE;

    #Busy := #reqActive AND #busyRaw;
END_FUNCTION_BLOCK

// -----------------------------------------------------------------------------
// FB_RecipePreScan - Pre-scan recipe for limit validation
// DOC:
//  purpose: Scan recipe lines before execution to compute bounding box and detect
//           any soft-limit violations. Runs in batches to avoid long PLC scan times.
//  inputs: Execute (rising edge), LineCount
//  outputs: Done, Valid, ErrorLine (first offending line), MinX/MaxX, MinZ/MaxZ
//  notes: Designed for non-blocking operation - processes N lines per PLC cycle.
// -----------------------------------------------------------------------------
FUNCTION_BLOCK "FB_RecipePreScan"
{ S7_Optimized_Access := 'TRUE' }
VERSION : 0.1
    VAR_INPUT
        Execute : Bool;             // Rising edge starts pre-scan (level input)
        LineCount : Int;            // Number of lines to scan
    END_VAR
    VAR_OUTPUT
        Done : Bool;                // TRUE when pre-scan finished
        Valid : Bool;               // TRUE if no limit violations found
        ErrorLine : Int := -1;      // Line with first error (-1 = none)
        ErrorDesc : String[60];     // Human-readable description of first violation
        MinX : Real;                // Computed bounding box minimum X
        MaxX : Real;                // Computed bounding box maximum X
        MinZ : Real;                // Computed bounding box minimum Z
        MaxZ : Real;                // Computed bounding box maximum Z
        Progress : Real;            // Pre-scan progress 0-100% for HMI display
    END_VAR
    VAR_IN_OUT
        // Bound to "DB_SelectedRecipe".Lines -- the work-memory buffer, never a
        // DB_RecipeProgram* (those are load-memory only). Must match that DB.
        // <<< GENERATED:PRESCAN_LINES -- do not hand-edit; run tools/gen_recipe_slots.py --lines N >>>
        Lines : Array[0..799] of "RecipeLine"; // Recipe lines storage (in/out DB reference)
        // <<< END GENERATED:PRESCAN_LINES >>>
    END_VAR
    VAR
        state : Int;                // Local state machine
        scanIndex : Int;            // Current scan index (next line to process)
        scanEndIndex : Int;         // End index for current batch
        rtExecute : Bool;           // Rising-edge start detection
        prevExecute : Bool;         // Previous execute level (for edge)
        // Temp vars for pre-scan checks (#4 feedrate/spindle, #5 tool mapping)
        spindleRPM : Real;          // Decoded spindle RPM from Param byte
        tmpToolCode : Int;          // Tool code from recipe Param
        mapIndex : Int;             // Tool mapping loop index
        mapFound : Bool;            // Tool mapping search result
        cylTarget : Real;           // reserved (ITEM-38 ruler range check removed -- BackSupport is full-stroke on this machine)
        // Zero-length CMD=2 check (2026-09-15). Previous motion line's programmed end point --
        // the same point FB_RecipeHandler holds in currX/currZ when it launches the next line.
        prevMotionValid : Bool;     // FALSE until the first motion line (its start is wherever the axes are)
        prevMotionX : Real;
        prevMotionZ : Real;
        segDX : Real;
        segDZ : Real;
    END_VAR
    CONST
        // Recipe format: RecipeLine.Param encodes spindle speed as RPM ÷ 10.
        // Range: 0–255 byte → 0–2550 RPM. Clamp to DB_Spindle.MaxSpeed at runtime.
        // See PLC_Recipe_Format_Spec.md CMD_SPINDLE_ON.
        SPINDLE_PARAM_TO_RPM : Real := 10.0;
    END_CONST
BEGIN
    // -------------------------------------------------------------------------
    // Rising edge detection -- start once when Execute level rises
    // -------------------------------------------------------------------------
    #rtExecute := #Execute AND NOT #prevExecute;
    #prevExecute := #Execute;

    // NOTE: PreScan processes 10 lines per PLC scan cycle to avoid long scan blocks.
    // This preserves CPU responsiveness.
    // ErrorLine: the first line with a limit violation -- helps operator locate the issue.

    CASE #state OF

        // -----------------------------------------------------------------
        // === STATE_IDLE (0) ===
        // -----------------------------------------------------------------
        0: // IDLE -- waiting for Execute rising edge
            #Done := FALSE;
            #Progress := 0.0;
            IF #rtExecute THEN
                #scanIndex := 0;
                #MinX := "DB_MachineConfig".SoftLimit_MaxX;
                #MaxX := "DB_MachineConfig".SoftLimit_MinX;
                #MinZ := "DB_MachineConfig".SoftLimit_MaxZ;
                #MaxZ := "DB_MachineConfig".SoftLimit_MinZ;
                #ErrorLine := -1;
                #Valid := TRUE;
                #prevMotionValid := FALSE;
                #state := 10;
            END_IF;

        // -----------------------------------------------------------------
        // === STATE_SCANNING (10) ===
        // -----------------------------------------------------------------
        10: // SCANNING -- 10 lines scanned per cycle (batch processing)
            // Bounding box updated and soft limit checked for each G0/G1 line.
            // Other commands (SpindleOn, ToolChange, Dwell, End) skipped -- contain no position.
            #scanEndIndex := #scanIndex + 9;
            IF #scanEndIndex > #LineCount - 1 THEN
                #scanEndIndex := #LineCount - 1;
            END_IF;

            FOR #scanIndex := #scanIndex TO #scanEndIndex DO
                // Only check motion commands (G0=0, G1=1, continuous G1=2) for bounding box and limits.
                // CMD=2 MUST be inside this test -- a continuous line left out would skip the
                // soft-limit check entirely.
                IF #Lines[#scanIndex].CMD <= 2 THEN
                    // Update bounding box
                    IF #Lines[#scanIndex].X < #MinX THEN #MinX := #Lines[#scanIndex].X; END_IF;
                    IF #Lines[#scanIndex].X > #MaxX THEN #MaxX := #Lines[#scanIndex].X; END_IF;
                    IF #Lines[#scanIndex].Z < #MinZ THEN #MinZ := #Lines[#scanIndex].Z; END_IF;
                    IF #Lines[#scanIndex].Z > #MaxZ THEN #MaxZ := #Lines[#scanIndex].Z; END_IF;

                    // Check limits -- records which axis/direction was violated
                    IF #Lines[#scanIndex].X < "DB_MachineConfig".SoftLimit_MinX THEN
                        IF #ErrorLine < 0 THEN
                            #ErrorLine := #scanIndex;
                            #ErrorDesc := CONCAT(IN1 := 'X below min (',
                                          IN2 := CONCAT(IN1 := REAL_TO_STRING("DB_MachineConfig".SoftLimit_MinX),
                                          IN2 := ')'));
                        END_IF;
                        #Valid := FALSE;
                    ELSIF #Lines[#scanIndex].X > "DB_MachineConfig".SoftLimit_MaxX THEN
                        IF #ErrorLine < 0 THEN
                            #ErrorLine := #scanIndex;
                            #ErrorDesc := CONCAT(IN1 := 'X above max (',
                                          IN2 := CONCAT(IN1 := REAL_TO_STRING("DB_MachineConfig".SoftLimit_MaxX),
                                          IN2 := ')'));
                        END_IF;
                        #Valid := FALSE;
                    ELSIF #Lines[#scanIndex].Z < "DB_MachineConfig".SoftLimit_MinZ THEN
                        IF #ErrorLine < 0 THEN
                            #ErrorLine := #scanIndex;
                            #ErrorDesc := CONCAT(IN1 := 'Z below min (',
                                          IN2 := CONCAT(IN1 := REAL_TO_STRING("DB_MachineConfig".SoftLimit_MinZ),
                                          IN2 := ')'));
                        END_IF;
                        #Valid := FALSE;
                    ELSIF #Lines[#scanIndex].Z > "DB_MachineConfig".SoftLimit_MaxZ THEN
                        IF #ErrorLine < 0 THEN
                            #ErrorLine := #scanIndex;
                            #ErrorDesc := CONCAT(IN1 := 'Z above max (',
                                          IN2 := CONCAT(IN1 := REAL_TO_STRING("DB_MachineConfig".SoftLimit_MaxZ),
                                          IN2 := ')'));
                        END_IF;
                        #Valid := FALSE;
                    END_IF;

                    // Zero-length continuous line (2026-09-15). A CMD=2 line that repeats the
                    // previous motion point is skipped by the handler's degenerate-line branch,
                    // READ -> EXEC -> READ, without ever reaching STATE_VEL_WAIT -- where Pause,
                    // run permission and the path-deviation guard live -- while the velocity
                    // command keeps the axes on the old heading. A chain of them is unsupervised
                    // for 2 scans per line. Refuse the recipe instead.
                    // Expression and 0.01 mm threshold are IDENTICAL to the handler's vmNLen test
                    // on purpose: same REAL arithmetic, so the two can never disagree on a line.
                    // Non-motion lines (markers, spindle, cylinder) do not move the point, exactly
                    // as they do not touch currX/currZ in the handler.
                    IF #Lines[#scanIndex].CMD = 2 AND #prevMotionValid THEN
                        #segDX := #Lines[#scanIndex].X - #prevMotionX;
                        #segDZ := #Lines[#scanIndex].Z - #prevMotionZ;
                        IF SQRT(#segDX * #segDX + #segDZ * #segDZ) <= 0.01 THEN
                            IF #ErrorLine < 0 THEN
                                #ErrorLine := #scanIndex;
                                #ErrorDesc := 'CMD=2 zero-length: repeats previous point';
                            END_IF;
                            #Valid := FALSE;
                        END_IF;
                    END_IF;
                    #prevMotionX := #Lines[#scanIndex].X;
                    #prevMotionZ := #Lines[#scanIndex].Z;
                    #prevMotionValid := TRUE;
                END_IF;

                // #4 -- Feedrate check: G1 F-value above MaxVelocity (mm/min → mm/s for comparison)
                // Continuous G1 (CMD=2) must carry a real feed. With F = 0 the handler runs a
                // motion line as a rapid, and velocity mode could never apply to it.
                IF #Lines[#scanIndex].CMD = 2 AND #Lines[#scanIndex].F <= 0 THEN
                    IF #ErrorLine < 0 THEN
                        #ErrorLine := #scanIndex;
                        #ErrorDesc := 'CMD=2 continuous G1 needs F > 0';
                    END_IF;
                    #Valid := FALSE;
                END_IF;

                IF (#Lines[#scanIndex].CMD = 1 OR #Lines[#scanIndex].CMD = 2) AND #Lines[#scanIndex].F > 0 THEN
                    IF INT_TO_REAL(#Lines[#scanIndex].F) / "DB_MachineConfig".FeedrateConvFactor > "DB_MachineConfig".MaxVelocity THEN
                        IF #ErrorLine < 0 THEN
                            #ErrorLine := #scanIndex;
                            #ErrorDesc := CONCAT(IN1 := 'F exceeds MaxVelocity (',
                                          IN2 := CONCAT(IN1 := REAL_TO_STRING("DB_MachineConfig".MaxVelocity * "DB_MachineConfig".FeedrateConvFactor),
                                          IN2 := ' mm/min)'));
                        END_IF;
                        #Valid := FALSE;
                    END_IF;
                END_IF;

                // #4 -- Spindle speed check: CMD_SPINDLE_ON Param*10 RPM vs DB_Spindle.MaxSpeed
                IF #Lines[#scanIndex].CMD = 20 THEN   // CMD_SPINDLE_ON
                    #spindleRPM := INT_TO_REAL(BYTE_TO_INT(#Lines[#scanIndex].Param)) * SPINDLE_PARAM_TO_RPM;
                    IF #spindleRPM > "DB_Spindle".MaxSpeed THEN
                        IF #ErrorLine < 0 THEN
                            #ErrorLine := #scanIndex;
                            #ErrorDesc := CONCAT(IN1 := 'Spindle RPM exceeds max (',
                                          IN2 := CONCAT(IN1 := REAL_TO_STRING("DB_Spindle".MaxSpeed),
                                          IN2 := ' RPM)'));
                        END_IF;
                        #Valid := FALSE;
                    END_IF;
                END_IF;

                // #5 -- Tool mapping check: CMD_TOOL_CHANGE Param must exist in ToolCode_List
                // Skip if Bypass_ToolAxis=TRUE -- runtime also skips tool changes on bypass machines
                IF #Lines[#scanIndex].CMD = 10 AND NOT "DB_MachineConfig".Bypass_ToolAxis THEN
                    #tmpToolCode := BYTE_TO_INT(#Lines[#scanIndex].Param);
                    #mapFound := FALSE;
                    FOR #mapIndex := 1 TO "DB_MachineConfig".ToolCount DO
                        IF "DB_ToolConfig".ToolCode_List[#mapIndex] = #tmpToolCode THEN
                            #mapFound := TRUE;
                        END_IF;
                    END_FOR;
                    IF NOT #mapFound THEN
                        IF #ErrorLine < 0 THEN
                            #ErrorLine := #scanIndex;
                            #ErrorDesc := CONCAT(IN1 := 'Tool code not mapped: T',
                                          IN2 := INT_TO_STRING(#tmpToolCode));
                        END_IF;
                        #Valid := FALSE;
                    END_IF;
                END_IF;


            END_FOR;

            // #13 -- Progress: updated each batch so HMI shows scanning progress
            IF #LineCount > 0 THEN
                #Progress := INT_TO_REAL(#scanIndex) / INT_TO_REAL(#LineCount) * 100.0;
            END_IF;

            // NOTE: FOR loop auto-increments #scanIndex, extra +1 removed

            IF #scanIndex >= #LineCount THEN
                #state := 99;
            END_IF;

        // -----------------------------------------------------------------
        // === STATE_DONE (99) ===
        // -----------------------------------------------------------------
        99: // DONE
            #Done := TRUE;
            #Progress := 100.0;
            IF NOT #Execute THEN
                #Done  := FALSE;  // Drop Done on the release scan so a stale TRUE
                                  // cannot be misread as a fresh result by the caller
                #state := 0;
            END_IF;
    END_CASE;
END_FUNCTION_BLOCK

// -----------------------------------------------------------------------------
// FB_RecipeHandler - Execute recipe program line by line
// DOC:
//  purpose: Main recipe execution engine. Reads Lines[] and issues axis/spindle/tool requests.
//  inputs: Start/Stop/Pause/Reset control signals, LineCount
//  outputs: Busy/Done/Error, CurrentLine, Tool/Spindle requests, ActiveFeedrate, Progress
//  notes: No string parsing; recipe lines are pre-parsed into RecipeLine UDTs stored in DBs.
//         Designed to be deterministic and yield frequently to PLC scan cycle.
// -----------------------------------------------------------------------------
FUNCTION_BLOCK "FB_RecipeHandler"
{ S7_Optimized_Access := 'TRUE' }
VERSION : 0.1
    VAR_INPUT
        Start : Bool;               // Rising-edge or level to start/continue execution
        Stop : Bool;                // Stop execution (controlled stop)
        bStartEdge : Bool;          // Rising edge from Panel_Start_A AND Panel_Start_B (for sheet load confirm)
        Pause : Bool;               // Pause execution (retain position)
        Reset : Bool;               // Reset to beginning (clear internal state)
        StartLine : Int := 0;       // First line to execute on next run (0 = beginning; use savedLineIndex for warm restart)
        LineCount : Int;            // Total lines in program
    END_VAR
    VAR_OUTPUT
        Busy : Bool;                // Execution in progress
        Done : Bool;                // Program complete
        Paused : Bool;              // Execution paused (SingleStep or Pause)
        Error : Bool;               // Error occurred
        ErrorID : Word;             // Error code (DB_ErrorCodes)
        CurrentLine : Int;          // Current line index being executed
        // Pass display (CMD_OP_MARK / CMD_PASS_MARK). 0 = no pass information:
        // either the recipe carries no markers, or execution has not reached the
        // first one yet. The HMI must blank the group on 0, not show "0 / 0".
        CurrentOp : Int;            // Operation number the current line belongs to
        TotalOps : Int;             // Operations in the program
        CurrentPass : Int;          // Pass number within the current operation
        TotalPasses : Int;          // Passes in the current operation
        ToolChangeReq : Bool;       // Tool change requested by recipe
        ToolReqNumber : Int;        // Requested tool number (from recipe Param)
        SpindleReqStart : Bool;     // Spindle start request flag
        SpindleReqStop : Bool;      // Spindle stop request flag
        SpindleReqSpeed : Real;     // Spindle speed request (RPM)
        ActiveFeedrate : Real;      // Current feedrate (mm/min) for HMI display
        Progress : Real;            // Progress percentage 0-100
    END_VAR
    VAR_IN_OUT
        // Bound to "DB_SelectedRecipe".Lines -- the work-memory buffer, never a
        // DB_RecipeProgram* (those are load-memory only). Must match that DB.
        // <<< GENERATED:HANDLER_LINES -- do not hand-edit; run tools/gen_recipe_slots.py --lines N >>>
        Lines : Array[0..799] of "RecipeLine"; // Reference to recipe lines in DB
        // <<< END GENERATED:HANDLER_LINES >>>
        Axis_X : TO_PositioningAxis;           // Axis TO IN_OUT
        Axis_Z : TO_PositioningAxis;
    END_VAR
    VAR
        state : Int;                // Internal state machine
        lineIndex : Int;           // Current executing line index

        // Current motion targets and feedback
        targX : Real;               // Target X for current line
        targZ : Real;               // Target Z for current line
        currX : Real;               // Current X tracked by handler
        currZ : Real;               // Current Z tracked by handler
        velX : Real;                // Velocity command for X (mm/s)
        velZ : Real;                // Velocity command for Z (mm/s)

        // Temporary calculation variables
        deltaX : Real;
        deltaZ : Real;
        totalDist : Real;
        feedrate : Real;            // Calculated feedrate (mm/s)
        // Tool mapping helpers
        tmpToolCode : Int;          // Raw tool code from recipe Param (e.g. 101)
        mapIndex : Int;             // Loop index for mapping lookup
        mapFound : Bool;            // TRUE if mapping found

        // Move control flags
        bTrigMove : Bool;           // Trigger movement this cycle
        bMoveX : Bool;              // X axis needs to move
        bMoveZ : Bool;              // Z axis needs to move
        bHaltTrig : Bool;           // Trigger halt (Stop)
        // Resume target after PAUSED -- STATE_PAUSE_RETURN (803) jumps here.
        // Every pause site sets it explicitly: a motion pause resumes via
        // STATE_READ (re-read the line endpoint, then EXEC recomputes the
        // remaining move), and the non-motion states (SPINDLE_WAIT / DWELL /
        // SPINDLE_STOP_WAIT / CYL_GOTO_WAIT) return to themselves -- resuming
        // those via STATE_EXEC executed a move to the non-motion line's X/Z
        // placeholders (0,0) and drove both axes to home.
        //
        // The default below is unreachable today: 803 is only entered through a
        // pause site and all five write this variable. It is STATE_READ and NOT
        // STATE_EXEC (2026-09-02) because STATE_EXEC is now hoisted out of the
        // CASE -- a resume landing on 20 would run EXEC in the same scan that
        // 803 clears bTrigMove, destroying the MC_MoveAbsolute Execute edge and
        // leaving the axis dead after Continue with no error raised. If a sixth
        // pause site is ever added and forgets to set this, STATE_READ fails
        // safe. Written as a literal because the CONST block is declared below.
        pauseReturnState : Int := 10;  // 10 = STATE_READ (safe default)
        // Pause-retract: interruption point captured on pause, returned to on resume.
        resumeX : Real;             // Interruption-point X (return target after retract)
        resumeZ : Real;             // Interruption-point Z

        // Motion FB instances used by handler
        fbMoveX : "FB_Axis_AbsPos";
        fbMoveZ : "FB_Axis_AbsPos";
        fbHaltX : "FB_Axis_Halt";
        fbHaltZ : "FB_Axis_Halt";

        // ---------------------------------------------------------------------
        // Velocity-mode continuous path (EXPERIMENTAL, branch exp/velocity-path-350)
        // ---------------------------------------------------------------------
        // Runs of CMD_LINEAR_CONT (CMD=2) lines are driven with MC_MoveVelocity
        // instead of MC_MoveAbsolute, so the axes do not stop at every recipe line.
        // Design, guards and test plan: docs/MotionSmoothing.md section 9.
        //
        // TWO instances per axis, used alternately (A, B, A, ...). MC_MoveVelocity
        // latches Velocity only on a rising edge of Execute; with one instance every
        // new segment would need an Execute-low scan first. Raising the OTHER
        // instance aborts the running one and applies the new vector in the same
        // scan. An instance is never raised twice in a row, so it always sees at
        // least one Execute-low scan before its next edge.
        //
        // MC_MoveVelocity does NOT stop when Execute drops. Every way out of this
        // mode other than the MC_MoveAbsolute hand-over must therefore halt the
        // axes: Pause/Stop/ERROR through bHaltTrig, Reset through vmHaltReq.
        mcVelXA : MC_MoveVelocity;
        mcVelXB : MC_MoveVelocity;
        mcVelZA : MC_MoveVelocity;
        mcVelZB : MC_MoveVelocity;
        vmActive    : Bool;         // A velocity command owns the axes right now
        vmUseB      : Bool;         // Which instance pair carries the live command
        vmHaltReq   : Bool;         // Reset left the axes moving -- hold MC_Halt until stopped
        vmEligible  : Bool;         // This line runs in velocity mode (computed in EXEC)
        vmWasActive : Bool;         // EXEC is handing a velocity run over to MC_MoveAbsolute
        vmErr       : Bool;         // Live instance pair reports Error (from last call)
        vmAborted   : Bool;         // Live instance pair was aborted by someone else
        vmMaxDev    : Real;         // VelPath_MaxDeviation clamped to VM_MAXDEV_MIN..VM_MAXDEV_MAX (mm), every scan
        vmVelX      : Real;         // Signed X velocity of the live segment (mm/s)
        vmVelZ      : Real;         // Signed Z velocity of the live segment (mm/s)
        vmDX        : Real;         // Launch vector, actual position -> line end (mm)
        vmDZ        : Real;
        vmDist      : Real;
        vmUX        : Real;         // Unit direction of the live segment
        vmUZ        : Real;
        vmSegLen    : Real;         // Length of the live segment at launch (mm)
        vmRem       : Real;         // Remaining distance along the segment (mm)
        vmLat       : Real;         // Distance off the segment line (mm)
        vmSwitchDist : Real;        // Remaining distance at which the next line takes over (mm)
        vmNDX       : Real;         // Programmed segment: previous programmed end point -> this line's end
        vmNDZ       : Real;
        vmNLen      : Real;
        vmAhead     : Real;         // How far this line's end point still is AHEAD of the axes, along the programmed segment (mm)
        vmNLat      : Real;         // Distance of the axes from the programmed segment line (mm)
        vmSkipDist  : Real;         // vmAhead at or below which the line counts as already passed (mm)
        vmLeadDist  : Real;         // Distance the axes cover in VelPath_LeadTime at the live commanded speed (mm)
        vmLoop      : Int;          // Same-scan catch-up loop counter
        vmNextOK    : Bool;         // Next line may itself run in velocity mode (catch-up may skip into it)
        vmUnsupScans : Int;         // Safety net 2: consecutive scans a velocity instance is Busy with no command live
        vmSkipCount : Int;          // Lines skipped by the catch-up loop in THIS scan
        vmBrakeV    : Real;         // Hand-over: live speed of the axis being evaluated (mm/s)
        vmBrakeX    : Real;         // Hand-over: X braking distance from its live speed, with margin (mm)
        vmBrakeZ    : Real;         // Hand-over: Z braking distance from its live speed, with margin (mm)
        actX        : Real;         // Axis ActualPosition snapshot
        actZ        : Real;

        // Timers for move timeout and dwell
        tonMoveTimeout : TON;
        tonPauseMove : TON;         // Timeout guard for pause retract/return moves
        tonDwell : TON;             // Dwell timer for CMD_DWELL
        tonAtSpeed : TON;           // Timeout timer for spindle at-speed wait (STATE_SPINDLE_WAIT)
        dwellTime : Time;           // Calculated dwell duration

        // Edge detection for Start/StepNext
        prevStart : Bool;           // previous Start level
        rtStart : Bool;             // rising edge Start
        prevStepNext : Bool;        // previous StepNext level
        rtStepNext : Bool;          // rising edge StepNext

        // Override temporary
        overridePercent : Real;     // Feedrate override percent (50..200)
    END_VAR

    CONST
        // Build tag. BUMP ON EVERY CHANGE TO THIS FB (date + letter). Check it by
        // opening this block ONLINE in TIA (the CONST section shows the CPU's copy),
        // or by an online/offline compare. Deliberately written nowhere: a DB field
        // would force a second block to be imported and downloaded.
        BUILD_TAG : String[16] := '2026-09-29c';

        STATE_IDLE : Int := 0;
        STATE_READ : Int := 10;
        STATE_EXEC : Int := 20;
        STATE_WAIT : Int := 30;
        STATE_TOOL_REQ : Int := 40;
        STATE_TOOL_WAIT : Int := 50;
        STATE_SPINDLE : Int := 55;   // Spindle command processing
        STATE_SPINDLE_WAIT : Int := 56;  // Wait for spindle AtSpeed after start command
        STATE_DWELL : Int := 57;     // Dwell/wait timer
        STATE_SPINDLE_STOP_WAIT : Int := 58;  // Wait for spindle to fully stop before proceeding
        STATE_NEXT : Int := 60;
        STATE_STEP_WAIT : Int := 65;  // Wait for StepNext in SingleStepMode
        STATE_CYL_GOTO      : Int := 70;   // CMD=40: set BackSupport TargetPos and trigger extend
        STATE_CYL_GOTO_WAIT : Int := 71;   // CMD=40: wait for BackSupport AtSetpoint or error
        STATE_VEL_WAIT      : Int := 32;   // Velocity-mode segment in progress (EXPERIMENTAL)
        VM_CATCHUP_MAX      : Int := 10;   // Most passed lines skipped in ONE scan (simulation needed 2 at T = 0.1 s)
        VM_MAXDEV_MIN       : Real := 0.05; // mm -- floor for the operator-set deviation limit (0 / negative / typo -> strict)
        VM_MAXDEV_MAX       : Real := 5.0;  // mm -- ceiling: a typo (30, 300) must not switch the path guard off.
                                            //       Raised from 1.0 to 5.0 on 2026-09-21 (user) -- 1.0 was the
                                            //       original default and the operator could not get past it.
                                            //       NOTE the meaning changes above 0.8 mm: the final-pass
                                            //       roller-mandrel gap IS the 0.8 mm sheet, so a limit set above
                                            //       it no longer protects the mandrel -- it only catches a
                                            //       runaway. Commission with the smallest value that runs.
        VM_UNSUPERVISED_SCANS : Int := 2;  // Safety net 2 grace: a hand-over MC_MoveAbsolute or MC_Halt aborts the
                                           // velocity command within ~1 scan; Busy on the 3rd scan = unsupervised
        // Hand-over speed floor: braking-distance test (2026-09-29, see STATE_EXEC).
        // COPIES of the X/Z TO dynamics -- keep in step with the TO (docs/MotionSmoothing.md
        // table at the top) and with tools/split_recipe_db.py HANDOVER_* constants.
        // Going stale is benign one way and bounded the other: a SHORTER real braking
        // distance (faster jerk, e.g. t1 0.03) floors a few more axes, error <= this
        // estimate; a LONGER one (t1 back to 0.3) can bring the old crawl back on a line.
        VM_HO_JERK   : Real := 2564.0;  // mm/s^3 -- TO jerk (acc/t1 = dec/t2, t1 0.06 s)
        VM_HO_DEC    : Real := 184.6;   // mm/s^2 -- TO deceleration
        VM_HO_SCAN   : Real := 0.045;   // s      -- OB1 cycle, measured 40-45 ms 2026-09-15
        VM_HO_MARGIN : Real := 2.0;     // covers servo following error and scan jitter the model ignores
        STATE_DONE : Int := 99;
        STATE_PAUSED : Int := 800;         // Pause entry: halt axes, then retract
        STATE_PAUSE_RETRACT : Int := 801;  // Moving to retracted (tool-clear) position
        STATE_PAUSE_HOLD    : Int := 802;  // Held at retracted position, waiting for Continue
        STATE_PAUSE_RETURN  : Int := 803;  // Moving back to interruption point before resume
        STATE_STOPPING : Int := 850;  // Halt triggered, waiting for axes to stop
        STATE_ERROR : Int := 999;

        CMD_RAPID : Byte := 0;
        CMD_LINEAR : Byte := 1;
        // EXPERIMENTAL (exp/velocity-path-350): G1 that MAY blend into the next line.
        // Per-line, not modal, so a warm restart or pause-resume from any line is
        // correct without scanning backwards. CMD=1 stays an exact stop, always.
        CMD_LINEAR_CONT : Byte := 2;
        CMD_TOOL_CHANGE : Byte := 10;
        CMD_SPINDLE_ON : Byte := 20;
        CMD_SPINDLE_OFF : Byte := 21;
        CMD_DWELL : Byte := 30;
        CMD_CYLINDER_GOTO : Byte := 40;     // BackSupport full extend (PositioningMode=0 on this machine; Param ignored)
        CMD_ATMO          : Byte := 41;     // BackSupport atmosphere. Param=1 → SolAtmo ON, Sol_A stays ON;
                                            // Param=2 → SolAtmo OFF + Cmd_Retract (Sol_A off, Sol_B on);
                                            // Param=3 → release retract, all coils off.
                                            // (The old "Sol_B+SolAtmo ON" at P1 was the SolB_Cmd41
                                            //  override, deleted 2026-08-07 -- see ITEM-41.)
        // Pass markers -- display only, no machine action. Emitted by SpinningCam
        // when its PLC-mode "pass markers" option is on; absent otherwise, and a
        // recipe without them runs exactly as before with the HMI fields blank.
        // The pass number is data SpinningCam already computes and used to throw
        // away in a source comment ("[Op1 P2]"), which the compiler discards.
        // See Program/docs/letter_spinningcam_pass_markers.md.
        CMD_OP_MARK   : Byte := 50;     // Param = operation number, F = total operations
        CMD_PASS_MARK : Byte := 51;     // Param = pass number in op, F = total passes in op
        CMD_END : Byte := 99;

        // Recipe format: RecipeLine.Param encodes spindle speed as RPM ÷ 10.
        // Range: 0–255 byte → 0–2550 RPM. Clamp to DB_Spindle.MaxSpeed at runtime.
        // See PLC_Recipe_Format_Spec.md CMD_SPINDLE_ON.
        SPINDLE_PARAM_TO_RPM : Real := 10.0;
    END_CONST
BEGIN
    // =========================================================================
    // FB_RecipeHandler -- Execution logic summary
    // =========================================================================
    // Called every PLC scan cycle.
    // State machine:
    //   IDLE(0) → READ(10) → EXEC(20) → WAIT(30) → NEXT(60) → READ(10) → ...
    //   Special branches: TOOL_REQ(40)→TOOL_WAIT(50), SPINDLE(55), DWELL(57),
    //                     STEP_WAIT(65), PAUSED(800), STOPPING(850), DONE(99), ERROR(999)
    //   Velocity mode (EXPERIMENTAL): READ(10) -> EXEC(20) -> VEL_WAIT(32) -> READ(10) ...
    //                     for runs of CMD=2 (continuous G1) lines; the last line of a run falls
    //                     back to EXEC -> WAIT(30) with MC_MoveAbsolute.
    // All axis moves are performed via fbMoveX / fbMoveZ.
    // Spindle and tool change requests are passed to FB_Process via flags (no direct drive access).
    // =========================================================================

    // Rising edge detection -- Start button
    #rtStart := #Start AND NOT #prevStart;
    #prevStart := #Start;

    // NOTE: prevStart is cleared on Reset -- consecutive starts are reliably detected.

    // SingleStep edge detection
    #rtStepNext := "DB_HMI".StepNext AND NOT #prevStepNext;
    #prevStepNext := "DB_HMI".StepNext;

    // -------------------------------------------------------------------------
    // RESET -- Rewind program to beginning, clear all flags
    // Can be applied while running; caller must stop axes first.
    // -------------------------------------------------------------------------
    IF #Reset THEN
        #lineIndex := #StartLine;   // 0 = normal start; >0 = warm restart from saved line
        #state := STATE_IDLE;
        #Error := FALSE;
        #ErrorID := 0;
        #Busy := FALSE;
        #Done := FALSE;
        #Paused := FALSE;
        #ToolChangeReq := FALSE;
        // Pass display back to "unknown". This is the only clear path they need:
        // FB_Process mirrors these to DB_HMI every scan, so zeroing here blanks
        // the HMI too -- see the mirror comment in 06_MainProcess.scl.
        #CurrentOp := 0;
        #TotalOps := 0;
        #CurrentPass := 0;
        #TotalPasses := 0;
        // BUG FIX: Clear internal flags so rising-edge detection works on next Start
        #prevStart := FALSE;
        #bTrigMove := FALSE;
        #bMoveX := FALSE;
        #bMoveZ := FALSE;
        #bHaltTrig := FALSE;
        // Velocity mode: dropping Execute does not stop MC_MoveVelocity, and IDLE
        // drives bHaltTrig FALSE -- so a reset taken mid-run latches its own halt.
        IF #vmActive THEN
            #vmHaltReq := TRUE;
        END_IF;
        #vmActive := FALSE;
        // Clear stale resume target from a previous pause. STATE_READ, not
        // STATE_EXEC -- see the declaration comment for why 20 is unsafe now
        // that STATE_EXEC is hoisted out of the CASE.
        #pauseReturnState := STATE_READ;
        #SpindleReqStart := FALSE;
        #SpindleReqStop := FALSE;
        // Reset timers -- no stale ET remains on next run
        #tonMoveTimeout(IN := FALSE, PT := "DB_MachineConfig".Timeout_Motion);
        #tonPauseMove(IN := FALSE, PT := "DB_MachineConfig".Timeout_Motion);
        #tonDwell(IN := FALSE, PT := T#0S);
        // Clear CMD=40/41 BackSupport commands so next run starts clean.
        // Cmd_Retract is cleared here too: it is latched by CMD=41 P2 and by the
        // end-of-recipe retract in FB_Process, and a recipe must never start with a
        // stale retract command still held. FB_Process drops its end-retract latch on
        // leaving STOPPED/ERROR/COMPLETE, so this cannot cut that sequence short.
        "DB_Cylinder_BackSupport".Cmd_Extend  := FALSE;
        "DB_Cylinder_BackSupport".Cmd_Retract := FALSE;
        "DB_Cylinder_BackSupport".SolAtmo_Cmd := FALSE;
    END_IF;

    // -------------------------------------------------------------------------
    // STOP -- Controlled, error-free stop sequence
    // Halt triggered → waits in STATE_STOPPING until both axes fully stop
    // → STATE_DONE. Error/ErrorID untouched (operator stop is not an error).
    // -------------------------------------------------------------------------
    IF #Stop AND #state <> STATE_IDLE AND #state <> STATE_ERROR
              AND #state <> STATE_STOPPING AND #state <> STATE_DONE THEN
        // User Stop = controlled, error-free stop
        // Safely interrupt moves using FB_Axis_Halt.
        // Waits in STATE_STOPPING until halt completes, then STATE_DONE.
        #bHaltTrig := TRUE;
        // Drop any active move trigger so the pending halt has sole control of the axes.
        // Required because the pause-retract states (801/803) leave bTrigMove TRUE;
        // without this, MC_MoveAbsolute and MC_Halt would fight on the same axis.
        #bTrigMove := FALSE;
        // Velocity mode: release the velocity command; bHaltTrig above stops the axes.
        #vmActive := FALSE;
        #Paused := FALSE;
        // Clear BackSupport Cmd_Extend -- if stop fires during CMD=40 (STATE_CYL_GOTO_WAIT),
        // without this the cylinder keeps extending through the entire stop/home sequence.
        "DB_Cylinder_BackSupport".Cmd_Extend := FALSE;
        #state := STATE_STOPPING;
    END_IF;

    // Velocity-path deviation limit (2026-09-16). OPERATOR-OWNED: DB_MachineConfig.
    // VelPath_MaxDeviation is set from the HMI and is no longer written by FC_LoadConfig.
    // Clamped here, once, and every guard reads #vmMaxDev -- never the raw config value,
    // so a mistyped 0 or 30 cannot make the guard fire constantly or never.
    #vmMaxDev := "DB_MachineConfig".VelPath_MaxDeviation;
    IF NOT (#vmMaxDev >= VM_MAXDEV_MIN) THEN      // also catches NaN
        #vmMaxDev := VM_MAXDEV_MIN;
    ELSIF #vmMaxDev > VM_MAXDEV_MAX THEN
        #vmMaxDev := VM_MAXDEV_MAX;
    END_IF;

    // Move timeout timer -- only counts during STATE_WAIT and STATE_VEL_WAIT.
    // PT is DB_MachineConfig.Timeout_Motion (T#300S as configured in FC_LoadConfig).
    // If the axis does not return Done within it, error 16#0008 (Motion Timeout) is raised.
    // Do NOT quote the figure in comments or operator strings -- it drifted once already:
    // three ErrorDetail strings said '(30s limit)' while the real value was 300 s (ITEM-56e).
    #tonMoveTimeout(IN := (#state = STATE_WAIT) OR (#state = STATE_VEL_WAIT), PT := "DB_MachineConfig".Timeout_Motion);

    // Pause retract/return move timeout -- counts only while a pause move is in progress.
    // Guards against a stuck axis hanging the machine in the retract or return phase.
    #tonPauseMove(IN := (#state = STATE_PAUSE_RETRACT OR #state = STATE_PAUSE_RETURN),
                  PT := "DB_MachineConfig".Timeout_Motion);

    // State machine
    CASE #state OF

        // -----------------------------------------------------------------
        // === STATE_IDLE (0) ===
        // -----------------------------------------------------------------
        0: // IDLE
            #Busy := FALSE;
            #Done := FALSE;
            #Paused := FALSE;
            #bTrigMove := FALSE;
            #bHaltTrig := FALSE;

            // NOT vmHaltReq: a reset taken during a velocity run is still braking;
            // starting a move now would fight that MC_Halt.
            IF #rtStart AND #LineCount > 0 AND NOT #vmHaltReq THEN
                #lineIndex := #StartLine;   // 0 = normal start; >0 = warm restart
                #currX := #Axis_X.ActualPosition;
                #currZ := #Axis_Z.ActualPosition;
                #Busy := TRUE;
                #state := STATE_READ;
            END_IF;

        // -----------------------------------------------------------------
        // === STATE_READ (10) ===
        // -----------------------------------------------------------------
        10: // READ - Read current line
            IF #lineIndex >= #LineCount THEN
                #state := STATE_DONE;
            ELSE
                // Read line data
                #targX := #Lines[#lineIndex].X;
                #targZ := #Lines[#lineIndex].Z;

                // Check command type
                CASE #Lines[#lineIndex].CMD OF
                    CMD_END:
                        #state := STATE_DONE;

                    CMD_TOOL_CHANGE:
                        // ITEM-35 (fixed 2026-08-16): on a bypassed machine, skip the line here --
                        // BEFORE the mapping lookup. FB_RecipePreScan already skips its tool-mapping
                        // check under the same flag, but the runtime skip used to live in FB_Process
                        // STATE_RUNNING (clearing ToolChangeReq), which is reached only AFTER this
                        // lookup has already raised 16#0308. So a bypass machine passed validation
                        // and then faulted mid-run on its first CMD=10 with an unmapped code.
                        // Same shape as the Bypass_Spindle branch below -- keep them consistent.
                        IF "DB_MachineConfig".Bypass_ToolAxis THEN
                            #state := STATE_NEXT;
                        ELSE
                            // Read raw tool code (supports post-processed codes like 101)
                            #tmpToolCode := BYTE_TO_INT(#Lines[#lineIndex].Param);
                            #mapFound := FALSE;
                            // Try explicit mapping in DB_ToolConfig.ToolCode_List
                            FOR #mapIndex := 1 TO "DB_MachineConfig".ToolCount DO
                                IF "DB_ToolConfig".ToolCode_List[#mapIndex] = #tmpToolCode THEN
                                    #ToolReqNumber := #mapIndex;
                                    #mapFound := TRUE;
                                END_IF;
                            END_FOR;
                            // If mapping not found -> report recipe tool number error (operator must map codes via HMI)
                            IF NOT #mapFound THEN
                                #ErrorID := 16#0308; // Recipe: Invalid tool number
                                "DB_Diagnostic".Error_Text := CONCAT(IN1 := 'Tool code ', IN2 := INT_TO_STRING(#tmpToolCode));
                                "DB_Diagnostic".Error_Line := #lineIndex;
                                "DB_Diagnostic".Error_Code := #ErrorID;
                                // Single-writer: HMI error comes from FB_AlarmManager (FB_Process forwards
                                // #ErrorID from STATE_RUNNING). The missing code number goes into ErrorDetail.
                                "DB_HMI".ErrorDetail    := CONCAT(IN1 := 'Tool code ', IN2 := CONCAT(
                                                           IN1 := INT_TO_STRING(#tmpToolCode),
                                                           IN2 := ' not mapped. Open Tool Setup, enter slot code & Apply.'));
                                #state := STATE_ERROR;
                            ELSE
                                // Mapping found -> request tool change for mapped slot
                                #state := STATE_TOOL_REQ;
                            END_IF;
                        END_IF;

                    CMD_SPINDLE_ON, CMD_SPINDLE_OFF:
                        IF "DB_HMI".Bypass_Spindle THEN
                            #state := STATE_NEXT;
                        ELSE
                            #state := STATE_SPINDLE;
                        END_IF;

                    CMD_DWELL:
                        // Dwell = wait for Param * 100ms
                        #dwellTime := INT_TO_TIME(BYTE_TO_INT(#Lines[#lineIndex].Param) * 100);
                        #tonDwell(IN := FALSE, PT := #dwellTime); // Reset timer
                        #state := STATE_DWELL;

                    CMD_CYLINDER_GOTO:
                        // BackSupport full extend -- waits AtSetpoint (Mode=0: after Timeout_Extend)
                        #state := STATE_CYL_GOTO;

                    CMD_ATMO:
                        // BackSupport atmosphere / retract control — fire-and-go (no axis wait).
                        // Operator spec 2026-08-07 (see DB_Cylinder_BackSupport header):
                        //   P1 -> atmosphere ON, Sol_A stays ON  (cylinder slack, still commanded out)
                        //   P2 -> atmosphere OFF, retract        (Sol_A off, Sol_B on)
                        //   P3 -> release retract                (all coils off, blocked centre holds)
                        //
                        // Sol_B is driven by the cylinder FB's own State 2, NOT by an output override.
                        // Cmd_Retract is a level input and nothing else writes it for this cylinder
                        // (FC_CylinderDispatch wires only the two *Full buttons), so a single write
                        // latches until we clear it at P3 or at end of recipe.
                        IF #Lines[#lineIndex].Param = 1 THEN
                            "DB_Cylinder_BackSupport".SolAtmo_Cmd := TRUE;   // energise atmosphere valve
                            // Sol_A deliberately left ON here (FB stays in State 3).
                        ELSIF #Lines[#lineIndex].Param = 2 THEN
                            "DB_Cylinder_BackSupport".SolAtmo_Cmd := FALSE;  // de-energise atmosphere valve
                            "DB_Cylinder_BackSupport".Cmd_Retract  := TRUE;  // FB State 3 -> 2: Sol_A off, Sol_B on
                        ELSIF #Lines[#lineIndex].Param = 3 THEN
                            "DB_Cylinder_BackSupport".SolAtmo_Cmd := FALSE;
                            "DB_Cylinder_BackSupport".Cmd_Retract  := FALSE; // FB State 2 -> 0: both coils off
                        END_IF;
                        #state := STATE_NEXT;

                    CMD_OP_MARK:
                        // Display only -- no actuator, no wait. Fire-and-go like CMD_ATMO.
                        #CurrentOp := BYTE_TO_INT(#Lines[#lineIndex].Param);
                        #TotalOps  := #Lines[#lineIndex].F;
                        // A new operation invalidates the previous operation's pass
                        // count. Without this, an op whose first pass marker is missing
                        // would keep showing the old op's "pass 10 of 10".
                        #CurrentPass := 0;
                        #TotalPasses := 0;
                        #state := STATE_NEXT;

                    CMD_PASS_MARK:
                        // Display only -- no actuator, no wait.
                        #CurrentPass := BYTE_TO_INT(#Lines[#lineIndex].Param);
                        #TotalPasses := #Lines[#lineIndex].F;
                        #state := STATE_NEXT;

                    CMD_RAPID, CMD_LINEAR, CMD_LINEAR_CONT:
                        #state := STATE_EXEC;

                    ELSE
                        // Unknown command - skip
                        #state := STATE_NEXT;
                END_CASE;
            END_IF;

        // -----------------------------------------------------------------
        // === STATE_WAIT (30) ===
        // -----------------------------------------------------------------
        30: // WAIT - Wait for motion complete
            #bTrigMove := FALSE;

            // Pause handling
            IF #Pause THEN
                #bHaltTrig := TRUE;
                // Resume via STATE_READ, not STATE_EXEC: the pause-retract states (800/802)
                // overwrite #targX/#targZ with retract/return geometry, destroying this line's
                // endpoint. STATE_READ re-reads the endpoint from #Lines[#lineIndex] before EXEC
                // recomputes the remaining move from currX/currZ (= interruption point after 803).
                // Going straight to EXEC computed deltaX = ABS(resumeX - resumeX) = 0 and silently
                // skipped the rest of the interrupted cut, jumping to the next line.
                #pauseReturnState := STATE_READ;  // motion pause: re-read endpoint, then recalc move
                #state := STATE_PAUSED;
            ELSE
                // Check completion based on which axes are moving
                IF (#bMoveX AND #bMoveZ) THEN
                    IF #fbMoveX.Done AND #fbMoveZ.Done THEN
                        #currX := #targX;
                        #currZ := #targZ;
                        #state := STATE_NEXT;
                    END_IF;
                ELSIF #bMoveX THEN
                    IF #fbMoveX.Done THEN
                        #currX := #targX;
                        #state := STATE_NEXT;
                    END_IF;
                ELSIF #bMoveZ THEN
                    IF #fbMoveZ.Done THEN
                        #currZ := #targZ;
                        #state := STATE_NEXT;
                    END_IF;
                ELSE
                    #state := STATE_NEXT;
                END_IF;

                // Error check -- TO/drive error or mechanical blockage
                // TO ErrorID: Siemens TO diagnostics code -- converted to readable text via FC_TO_ErrorText.
                // DB_Diagnostic.MoveX/Z_ErrorID: readable directly on HMI diagnostic page.
                IF (#bMoveX AND #fbMoveX.Error) OR (#bMoveZ AND #fbMoveZ.Error) THEN
                    IF #bMoveX AND #fbMoveX.Error THEN
                        #ErrorID := 16#0001;
                        "DB_Diagnostic".MoveX_ErrorID := #fbMoveX.ErrorID;
                        "DB_Diagnostic".TO_ErrorText  := "FC_TO_ErrorText"(Code := #fbMoveX.ErrorID);
                        "DB_Diagnostic".Error_Text := CONCAT(IN1 := 'X Move Failed: ', IN2 := "DB_Diagnostic".TO_ErrorText);
                        // Single-writer: HMI error from FB_AlarmManager (FB_Process forwards #ErrorID)
                        "DB_HMI".ErrorDetail    := CONCAT(IN1 := 'Ln:', IN2 := CONCAT(
                                                   IN1 := INT_TO_STRING(#lineIndex), IN2 := CONCAT(
                                                   IN1 := ' TO:', IN2 := "DB_Diagnostic".TO_ErrorText)));
                    ELSE
                        #ErrorID := 16#0002;
                        "DB_Diagnostic".MoveZ_ErrorID := #fbMoveZ.ErrorID;
                        "DB_Diagnostic".TO_ErrorText  := "FC_TO_ErrorText"(Code := #fbMoveZ.ErrorID);
                        "DB_Diagnostic".Error_Text := CONCAT(IN1 := 'Z Move Failed: ', IN2 := "DB_Diagnostic".TO_ErrorText);
                        // Single-writer: HMI error from FB_AlarmManager (FB_Process forwards #ErrorID)
                        "DB_HMI".ErrorDetail    := CONCAT(IN1 := 'Ln:', IN2 := CONCAT(
                                                   IN1 := INT_TO_STRING(#lineIndex), IN2 := CONCAT(
                                                   IN1 := ' TO:', IN2 := "DB_Diagnostic".TO_ErrorText)));
                    END_IF;
                    "DB_Diagnostic".Error_Line := #lineIndex;
                    "DB_Diagnostic".Error_Code := #ErrorID;
                    #state := STATE_ERROR;
                ELSIF #tonMoveTimeout.Q THEN
                    // Axis did not return Done within Timeout_Motion -- mechanical blockage, drive fault or TO issue
                    #ErrorID := 16#0008;
                    "DB_Diagnostic".Error_Line := #lineIndex;
                    "DB_Diagnostic".Error_Code := #ErrorID;
                    // Determine which axis is stuck (based on bMoveX/Z state).
                    // Single-writer: HMI error from FB_AlarmManager; axis goes into ErrorDetail.
                    IF #bMoveX AND #bMoveZ THEN
                        "DB_Diagnostic".Error_Text := 'Motion Timeout: X+Z axes';
                        "DB_HMI".ErrorDetail    := CONCAT(IN1 := 'X+Z no Done - Ln:',
                                                  IN2 := INT_TO_STRING(#lineIndex));
                    ELSIF #bMoveX THEN
                        "DB_Diagnostic".Error_Text := 'Motion Timeout: X axis';
                        "DB_HMI".ErrorDetail    := CONCAT(IN1 := 'X axis no Done - Ln:',
                                                  IN2 := INT_TO_STRING(#lineIndex));
                    ELSE
                        "DB_Diagnostic".Error_Text := 'Motion Timeout: Z axis';
                        "DB_HMI".ErrorDetail    := CONCAT(IN1 := 'Z axis no Done - Ln:',
                                                  IN2 := INT_TO_STRING(#lineIndex));
                    END_IF;
                    #state := STATE_ERROR;
                END_IF;

